Fanuc KAREL source: IO0031.KL

-- PROVISIONAL review KL for V940-1; original PC SHA256 ee4d76e11ce8cc25f1fd9313ae9302ff7b2241c482566ad424957239df7f1b54
-- Incomplete behavior may be omitted. Consult companion uncertainty JSON. Do not deploy.
PROGRAM IO0031
%NOLOCKGROUP
-- UNRESOLVED_LOCAL_POOL 5 cells at code offset 13; source declarations unknown
-- DIRECT_LOCAL_WORD_ACCESS alone does not prove INTEGER, REAL, or BOOLEAN
BEGIN
  -- V9_ZERO_TABLE_METADATA_HINT layout=0001; no indexed target words; source/name/runtime held
  -- V9_ZERO_GLOBAL_LAYOUT_HINT count-one $GROUP table, zero relocation slots, two routine descriptors; executable preamble and source held
  -- UNRESOLVED_PC offsets 0-18; opcodes 2B,2C,7B
  -- UNRESOLVED_PC offsets 23-30; opcodes 9D,23
  -- UNRESOLVED_PC offsets 35-49; opcodes 2E,22,9D,33,35
  -- UNRESOLVED_PC offsets 54-61; opcodes 9D,23
  -- UNRESOLVED_PC offsets 66-77; opcodes 2E,23
  -- UNRESOLVED_PC offsets 82-93; opcodes 9D,21,9D,52,1A
  -- UNRESOLVED_PC offsets 98-102; opcodes 7F
  -- UNRESOLVED_PC offsets 107-111; opcodes 27,AA
  -- UNRESOLVED_PC offsets 116-120; opcodes 7F
END IO0031
